Fanuc KAREL source: CE0056.KL

-- PROVISIONAL review KL for V1013-1; original PC SHA256 0422da9b2745e12c774bffa68d0dd93b2de92c661dee421b4be3529791cbd462
-- Incomplete behavior may be omitted. Consult companion uncertainty JSON. Do not deploy.
PROGRAM CE0056
%NOLOCKGROUP
-- UNRESOLVED_LOCAL_POOL 6 cells at code offset 94; source declarations unknown
-- DIRECT_LOCAL_WORD_ACCESS alone does not prove INTEGER, REAL, or BOOLEAN
BEGIN
  -- UNRESOLVED_PC offsets 0-1; opcodes 7B
  -- UNRESOLVED_PC offsets 6-16; opcodes 2D,7F
  -- UNRESOLVED_PC offsets 21-26; opcodes 7F,7B
  -- UNRESOLVED_PC offsets 31-43; opcodes 2D,9D,52,7F
  -- UNRESOLVED_PC offsets 48-53; opcodes 7F,7B
  -- UNRESOLVED_PC offsets 58-74; opcodes 2D,2E,69,7F
  -- UNRESOLVED_PC offsets 79-99; opcodes 7F,2B,2C,7B
  -- UNRESOLVED_PC offsets 104-115; opcodes 2E,23
  -- UNRESOLVED_PC offsets 120-131; opcodes 2E,23
  -- UNRESOLVED_PC offsets 136-147; opcodes 2E,23
  -- UNRESOLVED_PC offsets 152-163; opcodes 2E,23
  -- UNRESOLVED_PC offsets 168-175; opcodes 9D,23
  -- UNRESOLVED_PC offsets 180-187; opcodes 9C,23
  -- UNRESOLVED_PC offsets 192-202; opcodes 3F,75
  -- UNRESOLVED_PC offsets 207-217; opcodes 3F,75
  -- UNRESOLVED_PC offsets 222-236; opcodes 2E,22,9D,33,35
  -- UNRESOLVED_PC offsets 241-259; opcodes 2E,22,2E,33,35
  -- UNRESOLVED_PC offsets 264-290; opcodes 21,9D,52,21,2E,54,58,79
  -- UNRESOLVED_PC offsets 295-309; opcodes 21,9D,52,23
  -- UNRESOLVED_PC offsets 314-319; opcodes 7A
  -- UNRESOLVED_PC offsets 324-342; opcodes 21,2E,52,23
  -- UNRESOLVED_PC offsets 352-356; opcodes 7F
  -- UNRESOLVED_PC offsets 361-365; opcodes 27,AA
  -- UNRESOLVED_PC offsets 370-374; opcodes 7F
END CE0056
